// TIA Portal V17 export
// export: Created 2022-07-28T18:02:49.5126461Z, ExportSetting None, DisplayName Totally Integrated Automation Portal, DisplayVersion V17, DisplayName TIA Portal Openness, DisplayVersion V17, DisplayName TIA Portal Teamcenter Gateway, DisplayVersion V17, DisplayName TIA Portal Version Control Interface, DisplayVersion V17, DisplayName TIA Portal Test Suite Advanced, DisplayVersion V17, DisplayName SINAMICS Startdrive Advanced, DisplayVersion V17, DisplayName SINAMICS DCC, DisplayVersion V17, DisplayName SINAMICS Startdrive G130, G150, S120, S150, SINAMICS MV, S210, DisplayVersion V17, DisplayName SINAMICS Startdrive G110M, G120, G120C, G120D, G120P, G115D, DisplayVersion V17, DisplayName STEP 7 Professional, DisplayVersion V17, DisplayName SIMATIC Energy Suite, DisplayVersion V17, DisplayName STEP 7 CFC, DisplayVersion V17, DisplayName STEP 7 Safety, DisplayVersion V17, DisplayName WinCC Advanced / Unified PC, DisplayVersion V17, DisplayName SIMATIC Visualization Architect, DisplayVersion V17
FUNCTION "Lib_FC_PID_Cascad_AddNextPID" : Int   // FC26, SCL
{ S7_Optimized_Access := 'TRUE' }
// stored: SetENOAutomatically false
   VAR_IN_OUT
      i_InputArr : "_PID_Cascad_AutoCtrlPumpsAll";
   END_VAR
   VAR_TEMP
      t_ExistFree : Bool;
      ti_Cnt : Int;
      ti_CurrPID : Int;
   END_VAR
BEGIN
   //Set next available element for PID and reset all unavailable
   //Reset flags
   #t_ExistFree := false;
   #ti_CurrPID := -1;
   FOR #ti_Cnt := 0 TO 2 DO

       IF NOT #i_InputArr.Arr[#ti_Cnt].AutoControl_P.StatusGen.StartFull
           AND NOT #i_InputArr.Arr[#ti_Cnt].AutoControl_P.StatusGen.StartPID
           AND #i_InputArr.Arr[#ti_Cnt].Enabled
           AND #i_InputArr.Arr[#ti_Cnt].AutoControl_P.Mode.Auto
           AND #i_InputArr.Arr[#ti_Cnt].AutoControl_P.StatusGen.Ready
       THEN
           #t_ExistFree := true;
       END_IF;

       IF #i_InputArr.Arr[#ti_Cnt].AutoControl_P.StatusGen.StartPID
       THEN
           #ti_CurrPID := #ti_Cnt;
       END_IF;
   END_FOR;
   #Lib_FC_PID_Cascad_AddNextPID := #ti_CurrPID;

   //Set first free element
   IF #t_ExistFree
   THEN
       IF #ti_CurrPID >= 0
       THEN
           #i_InputArr.Arr[#ti_CurrPID].AutoControl_P.StatusGen.StartPID := false;
           #i_InputArr.Arr[#ti_CurrPID].AutoControl_P.StatusGen.StartFull := true;
       END_IF;

       FOR #ti_Cnt := 0 TO 2 DO
           IF NOT #i_InputArr.Arr[#ti_Cnt].AutoControl_P.StatusGen.StartFull
               AND NOT #i_InputArr.Arr[#ti_Cnt].AutoControl_P.StatusGen.StartPID
               AND #i_InputArr.Arr[#ti_Cnt].Enabled
               AND #i_InputArr.Arr[#ti_Cnt].AutoControl_P.Mode.Auto
               AND #i_InputArr.Arr[#ti_Cnt].AutoControl_P.StatusGen.Ready
           THEN
               #i_InputArr.Arr[#ti_Cnt].AutoControl_P.StatusGen.StartPID := true;
               #Lib_FC_PID_Cascad_AddNextPID := #ti_Cnt;
               RETURN;
           END_IF;
       END_FOR;

   END_IF;
END_FUNCTION
